Staubli VAL3: _WatchDog.pgx

public program _WatchDog()
  local bool l_bConnected
begin
  while true

    bIspower=isPowered()
    bIsEstop=(esStatus()==2)
//    if abs(herej()-data:jJhome)<{2,2,2,2,2,2}
//      data:bHome=true
//    else
//      data:bHome=false
//    endIf

    //检查通信状况
    nWorkingMode=workingMode(nWorkingStatus)
    call checkIoBus(l_bConnected)
    bConnected_Plc=l_bConnected
    delay(0)
  endWhile
end
